FUNCTION UINT_TO_ZEROSTRING : T_MAXSTRING
VAR_INPUT
	input : UDINT;
END_VAR
VAR
	tempString : T_MAXSTRING;
END_VAR

tempString := TO_STRING(input);
WHILE LEN(tempString) < 4 DO
	tempString := INSERT(tempString, '0', 0);
END_WHILE
UINT_TO_ZEROSTRING := tempString;

END_FUNCTION

(* stored: Version 1.1.0.1, ProductVersion 3.1.4024.12
   POU UINT_TO_ZEROSTRING: Id {014cd159-375b-4b71-a396-27af5aaf6299}, SpecialFunc None *)
